Fanuc KAREL source: ko00079.KL

PROGRAM KO00079
%STACKSIZE=65535
%PRIORITY=65535
%NOLOCKGROUP
VAR
P1 : XYZWPREXT
P2 : JOINTPOS9
F : BOOLEAN
OUT : XYZWPREXT
BEGIN
F=TRUE
-- UNSAFE_SOURCE_IR line 11: OUT = MIRROR(P1, convert_jointpos9_to_position(P2), F)
END KO00079
